% RSLogix 500 project I2P-JOB-06 DUNCAN_SUTTON.RSS, saved by version 10.00.00.00 %
PROJECT "ML01A"    % processor: Bul.1763 MicroLogix 1100 Series B %

PROGRAM FILES
  LAD 2   5 rungs

DATA FILES
  O0 OUTPUT  4 elements
  I1 INPUT  6 elements
  S2 STATUS  66 elements
  B3 BINARY  1 elements
  T4 TIMER  1 elements
  C5 COUNTER  1 elements
  R6 CONTROL  1 elements
  N7 INTEGER  1 elements
  F8 FLOAT  1 elements

LADDER 2
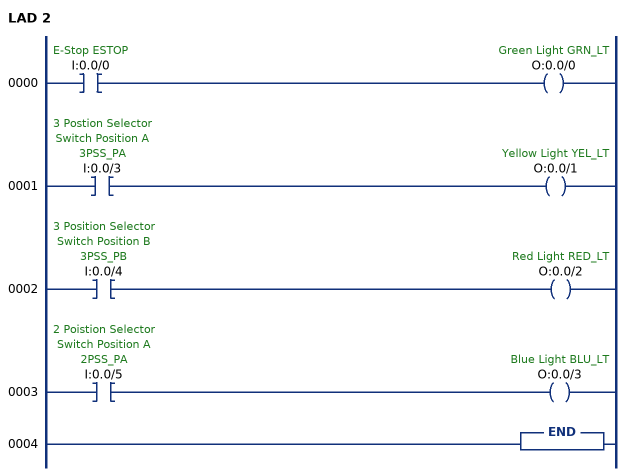
% Rung: 0 %
SOR XIC I:0.0/0 OTE O:0.0/0 EOR
%   I:0.0/0  ESTOP  "E-Stop" %
%   O:0.0/0  GRN_LT  "Green Light" %
% Rung: 1 %
SOR XIC I:0.0/3 OTE O:0.0/1 EOR
%   I:0.0/3  3PSS_PA  "3 Postion Selector Switch Position A" %
%   O:0.0/1  YEL_LT  "Yellow Light" %
% Rung: 2 %
SOR XIC I:0.0/4 OTE O:0.0/2 EOR
%   I:0.0/4  3PSS_PB  "3 Position Selector Switch Position B" %
%   O:0.0/2  RED_LT  "Red Light" %
% Rung: 3 %
SOR XIC I:0.0/5 OTE O:0.0/3 EOR
%   I:0.0/5  2PSS_PA  "2 Poistion Selector Switch Position A" %
%   O:0.0/3  BLU_LT  "Blue Light" %
% Rung: 4 %
SOR END EOR

OTHER DOCUMENTED ADDRESSES
  I:0.0/1  CR1_C  "Control Relay 1 Contact"
  I:0.0/2  CR2_C  "Control Relay 2 Contact"
  I:0.0/6  PB_1  "Pushbutton 1"
  I:0.0/7  PB_2  "Pushbutton 2"
  I:0.0/8  PB_3  "Pushbutton 3"
  O:0.0/4  CR_1  "Control Relay 1"
  O:0.0/5  CR_2  "Control Relay 2"
